{attribute 'GeneratedUsingTerminal: EL2522-0000-0017'}
{attribute addProperty BoxType "EL2522-0000-0017"}
{attribute addProperty Id "ControlAT %Q*Control_A8DDCD822Set_counter_valueAT %Q*UDINT4"}
{attribute addProperty CRC "1751890396"}
{attribute addProperty Size "6"}
TYPE ENC_Control_Channel_686BB9DC :
STRUCT
	{attribute addProperty Name "Control"}
	Control AT %Q* : Control_A8DDCD82;
	{attribute addProperty Name "Set_counter_value"}
	Set_counter_value AT %Q* : UDINT;
END_STRUCT
END_TYPE

(* stored: Version 1.2.0.0, ProductVersion 3.1.4024.9
   DUT ENC_Control_Channel_686BB9DC: Id {a9b3bc7b-ae2f-4d5d-9a92-21106121f688} *)
